// §3.8b — save the current parametrization as a named set.
//
// The set is a PROJECTION of the same deterministic walk that builds the
// §3.10.2 manifest: M_AppendConfig runs exactly as a QUERY_CONFIG would run it,
// and the pager files every capability of the requested ConfigKind as a
// (Scope, WriteKey) record. There is no second enumeration of "what this
// station's configuration consists of" to drift from the first (§1.1 O9).
//
// Kind selects which of the two kinds of set this is: STATION_CFG for a station
// set (deployment data), PAR_CFG for a model set (one model's recipe data).
METHOD SaveConfigSet : BOOL
VAR_INPUT
    SetName : STRING(80);
    Kind    : E_ConfigKind;
END_VAR
VAR
    info    : ST_ConfigSetInfo;
    records : INT;
END_VAR
SaveConfigSet := FALSE;
ConfigPersist.LastSetName := SetName;
ConfigPersist.LastSetRecords := 0;
IF NOT _M_SetOpAllowed() THEN
    RETURN;
END_IF
IF SetName = '' THEN
    RETURN;
END_IF
info.Used := TRUE;
info.SetName := SetName;
info.RootIdentity := Status.Name;
info.SetSchema := CONFIG_SET_SCHEMA;
info.ConfigRev := ConfigRev;
info.Kind := Kind;
IF Kind = E_ConfigKind.PAR_CFG THEN
    info.ModelCode := Model.ModelCode;     // a model set belongs to ONE model
ELSE
    info.ModelCode := '';
END_IF
info.RecordCount := 0;
info.CreatedAt := F_Now();
info.TimeSynchronized := F_TimeSynchronized();
IF NOT _configPager.M_SetupSetSave(Store := _configStore, Info := info) THEN
    RETURN;
END_IF
M_AppendConfig(Pager := _configPager);     // the SAME walk as the manifest
SaveConfigSet := _configPager.M_FinishSetSave(Records => records);
ConfigPersist.LastSetRecords := records;
IF SaveConfigSet THEN
    // The set now lives in the store's retained memory, which is not durable
    // until it is written out - the same promise as any other accepted write.
    _M_MarkPersistPending();
END_IF
END_METHOD

// §3.8b — apply a named set. STAGED and ALL-OR-NOTHING.
//
// Pass 1 validates every record through its owning module's typed handler and
// changes nothing. Only if all of them pass does pass 2 apply them. A
// half-applied machine parametrization is never a valid outcome, and the only
// way to guarantee that is to know the answer for every record before touching
// the first one.
//
// A record whose capability no longer exists fails pass 1 like any other and is
// REPORTED by name - never silently dropped, because a set that quietly skipped
// the one value that mattered restores a machine to almost its commissioned
// state, which is the failure that is hardest to notice.
METHOD LoadConfigSet : BOOL
VAR_INPUT
    SetName : STRING(80);
END_VAR
VAR
    info    : ST_ConfigSetInfo;
    record  : ST_ConfigRecord;
    i       : INT;
    applied : BOOL;
END_VAR
LoadConfigSet := FALSE;
ConfigPersist.LastSetName := SetName;
ConfigPersist.LastSetRecords := 0;
ConfigPersist.LastRejectScope := '';
ConfigPersist.LastRejectKey := '';
IF NOT _M_SetOpAllowed() THEN
    RETURN;
END_IF
IF NOT _configStore.M_ReadInfo(SetName := SetName, Info := info) THEN
    _M_RejectConfigSet(Scope := '', Key := SetName);
    RETURN;
END_IF
IF info.RootIdentity <> Status.Name THEN
    // The set carries the identity of the root that produced it precisely so
    // this can be asked. Every record's Scope is prefixed by that identity, so
    // a mismatch would fail record by record anyway - naming the root instead
    // tells the operator WHY in one line.
    _M_RejectConfigSet(Scope := info.RootIdentity, Key := '');
    RETURN;
END_IF
IF info.Kind = E_ConfigKind.PAR_CFG THEN
    // §3.8b: a MODEL set "shall be applied through the §3.8 changeover
    // transaction (PrepareRecipe -> recursive readiness -> infallible
    // CommitRecipe), never as a sequence of per-field writes". Applying it here
    // would be exactly that forbidden sequence, so it is refused. Saving a
    // model set is supported; loading one is a changeover this build does not
    // implement, and refusing is the honest half of that.
    _M_RejectConfigSet(Scope := info.ModelCode, Key := '');
    RETURN;
END_IF
// ---- pass 1: stage. Nothing in the machine changes in this loop. ----
FOR i := 1 TO info.RecordCount DO
    IF NOT _configStore.M_ReadRecord(SetName := SetName, Index := i,
            Record := record) THEN
        _M_RejectConfigSet(Scope := '', Key := SetName);
        RETURN;
    END_IF
    // §3.8d(e) - CONFIG_SET alone cannot replace a value this session could
    // not edit one at a time. Checked in the staging pass, so nothing moved.
    IF NOT Access.M_PermitsLevelLogged(Required := _M_DataLevelOf(TargetPath := record.Scope,
            WriteKey := record.WriteKey, ForWrite := TRUE)) THEN
        _M_RejectConfigSet(Scope := record.Scope, Key := record.WriteKey);
        RETURN;
    END_IF
    IF NOT _M_StageOneRecord(Record := record) THEN
        _M_RejectConfigSet(Scope := record.Scope, Key := record.WriteKey);
        RETURN;
    END_IF
END_FOR
// ---- pass 2: apply. Every record already proved acceptable on the SAME
// validator, so a refusal here cannot be a data problem. ----
FOR i := 1 TO info.RecordCount DO
    IF NOT _configStore.M_ReadRecord(SetName := SetName, Index := i,
            Record := record) THEN
        _M_ConfigSetHalfApplied(Scope := record.Scope, Key := record.WriteKey);
        RETURN;
    END_IF
    applied := _M_WriteBaseConfig(TargetPath := record.Scope,
        WriteKey := record.WriteKey, Revision := record.Revision,
        TextValue := record.ValueText, Commit := TRUE);
    IF NOT applied THEN
        applied := M_ApplyConfigWrite(Scope := record.Scope,
            WriteKey := record.WriteKey, Revision := record.Revision,
            TextValue := record.ValueText,
            RootReady := (_exec = E_ExecState.READY));
    END_IF
    IF NOT applied THEN
        _M_ConfigSetHalfApplied(Scope := record.Scope, Key := record.WriteKey);
        RETURN;
    END_IF
END_FOR
ConfigRev := ConfigRev + 1;
ConfigPersist.LastSetRecords := info.RecordCount;
_M_MarkPersistPending();
_M_RaiseMaintenance(Reason := E_Reason.EVENT_CONFIG_SET_APPLIED,
    Text := 'std.audit.configSetApplied');
LoadConfigSet := TRUE;
END_METHOD

// §3.8b — would this record be accepted? The same two-step the write path
// takes: framework-owned keys first, then the recursive walk to the owning
// module. Sharing the writers' own code with Commit := FALSE is what makes
// "staged" mean something: a separate validator could pass a record the write
// path would then refuse, and the load would be half-applied after all.
METHOD PRIVATE _M_StageOneRecord : BOOL
VAR_INPUT
    Record : ST_ConfigRecord;
END_VAR
_M_StageOneRecord := _M_WriteBaseConfig(TargetPath := Record.Scope,
    WriteKey := Record.WriteKey, Revision := Record.Revision,
    TextValue := Record.ValueText, Commit := FALSE);
IF _M_StageOneRecord THEN
    RETURN;
END_IF
_M_StageOneRecord := M_StageConfigWrite(Scope := Record.Scope,
    WriteKey := Record.WriteKey, Revision := Record.Revision,
    TextValue := Record.ValueText,
    RootReady := (_exec = E_ExecState.READY));
END_METHOD

// §3.8b — a record passed staging and then failed to apply. This cannot
// happen: both run the same validator on the same data in the same scan. If it
// ever does, the machine is half-parametrized and that is a state the standard
// says is never valid - so it is escalated as a BLOCKING alarm rather than
// returned as a FALSE somebody might retry. A framework defect that leaves a
// machine half-configured has to stop it, not inconvenience it.
METHOD PRIVATE _M_ConfigSetHalfApplied
VAR_INPUT
    Scope : STRING(80);
    Key   : STRING(160);
END_VAR
ConfigPersist.LastRejectScope := Scope;
ConfigPersist.LastRejectKey := Key;
AlarmLog.Raise(Reason := E_Reason.CONFIG_SET_REJECTED,
    Text := 'std.error.configSetHalfApplied', Source := Scope,
    Severity := E_Severity.HIGH, Category := E_Category.SYSTEM,
    ResetClass := E_ResetClass.MANUAL_RESET);
END_METHOD

// §3.8b — refresh the published listing of stored sets. Read-only, so it is
// gated on CONFIG_SET without the audited write path: seeing which sets exist
// is not replacing a machine's parametrization.
METHOD ListConfigSets : BOOL
VAR
    i     : INT;
    total : INT;
END_VAR
ListConfigSets := FALSE;
FOR i := 1 TO PL_Fraktal.MAX_CONFIG_SETS DO
    ConfigSets[i].Used := FALSE;
    ConfigSets[i].SetName := '';
    ConfigSets[i].RecordCount := 0;
END_FOR
ConfigSetCount := 0;
IF NOT Access.Permits(Gate := E_GatedAction.CONFIG_SET) THEN
    RETURN;
END_IF
IF _configStore = 0 THEN
    RETURN;
END_IF
total := _configStore.M_Count();
FOR i := 1 TO PL_Fraktal.MAX_CONFIG_SETS DO
    IF i > total THEN
        EXIT;
    END_IF
    IF _configStore.M_InfoAt(Index := i, Info := ConfigSets[i]) THEN
        ConfigSetCount := i;
    END_IF
END_FOR
ListConfigSets := TRUE;
END_METHOD

// §3.8b — serve one line of a set's JSON document. Line 0 is the header and
// 1..RecordCount are the records, so a client pulls a movable document a line
// at a time and no full document buffer ever exists in the PLC - the same
// paging discipline QUERY_CONFIG already uses for the manifest.
//
// This is what makes a set MOVABLE, which is the point of naming sets at all: a
// station's commissioning can leave the controller as text, be reviewed,
// diffed, version-controlled and put on the next machine.
METHOD ExportConfigSetLine : BOOL
VAR_INPUT
    SetName : STRING(80);
    Line    : INT;
END_VAR
VAR
    info   : ST_ConfigSetInfo;
    record : ST_ConfigRecord;
END_VAR
ExportConfigSetLine := FALSE;
ConfigSetDocument := '';
ConfigSetDocumentLine := Line;
ConfigSetDocumentLines := 0;
IF NOT Access.Permits(Gate := E_GatedAction.CONFIG_SET) THEN
    RETURN;
END_IF
IF _configStore = 0 THEN
    RETURN;
END_IF
IF NOT _configStore.M_ReadInfo(SetName := SetName, Info := info) THEN
    RETURN;
END_IF
ConfigSetDocumentLines := info.RecordCount;
IF Line <= 0 THEN
    ConfigSetDocument := _setJson.M_Header(Info := info);
ELSE
    IF NOT _configStore.M_ReadRecord(SetName := SetName, Index := Line,
            Record := record) THEN
        RETURN;
    END_IF
    IF NOT Access.M_PermitsLevel(Required := _M_DataLevelOf(TargetPath := record.Scope,
            WriteKey := record.WriteKey, ForWrite := FALSE)) THEN
        RETURN;                           // §3.8d(e): the export fails, it is not thinned
    END_IF
    ConfigSetDocument := _setJson.M_Record(Record := record);
END_IF
// An empty line means the projection REFUSED to render it rather than shorten
// it, so the export fails here instead of shipping a document with a hole.
ExportConfigSetLine := (ConfigSetDocument <> '');
END_METHOD

// §3.8b — take one line of a set's JSON document back in. A header line opens
// a store save, record lines append to it, and Commit closes it.
//
// Import writes into the STORE, never into the machine. Bringing a document in
// and applying it to the equipment are two decisions, and keeping them apart is
// what lets LoadConfigSet stay staged and all-or-nothing: an imported set is
// validated against THIS machine's capabilities when somebody chooses to load
// it, not silently as it arrives.
//
// Everything here is untrusted input in the fullest sense - hand-edited, from
// another vendor's tool, from another machine - so the line is parsed into a
// typed record and nothing more is assumed about it (§5.6, §14).
METHOD ImportConfigSetLine : BOOL
VAR_INPUT
    Line   : STRING(480);
    Commit : BOOL;
END_VAR
VAR
    info   : ST_ConfigSetInfo;
    record : ST_ConfigRecord;
END_VAR
ImportConfigSetLine := FALSE;
IF NOT _M_SetOpAllowed() THEN
    _importOpen := FALSE;
    RETURN;
END_IF
IF _setJson.M_ParseHeader(Line := Line, Info := info) THEN
    _importOpen := FALSE;
    info.Used := TRUE;
    info.RecordCount := 0;
    IF NOT _configStore.M_SaveBegin(Info := info) THEN
        RETURN;
    END_IF
    _importOpen := TRUE;
    ConfigPersist.LastSetName := info.SetName;
    ImportConfigSetLine := TRUE;
    RETURN;
END_IF
IF NOT _importOpen THEN
    RETURN;                                // a record before its header: refuse
END_IF
IF _setJson.M_ParseRecord(Line := Line, Record := record) THEN
    ImportConfigSetLine := _configStore.M_SaveRecord(Record := record);
    IF NOT ImportConfigSetLine THEN
        _configStore.M_SaveAbort();
        _importOpen := FALSE;
        RETURN;
    END_IF
ELSIF NOT Commit THEN
    // Neither a header nor a record, and not the closing call: the document is
    // not one this build understands. Abort rather than commit a partial set.
    _configStore.M_SaveAbort();
    _importOpen := FALSE;
    RETURN;
END_IF
IF Commit THEN
    ImportConfigSetLine := _configStore.M_SaveCommit();
    _importOpen := FALSE;
    IF ImportConfigSetLine THEN
        _M_MarkPersistPending();
    END_IF
END_IF
END_METHOD

// §3.8b - take part of a set line. A request carries at most 255 characters
// and an exported line may hold 480, so a longer line arrives as pieces:
// More = TRUE holds this piece and waits for the next; the first piece without
// More completes the line, which is then imported exactly like a whole one.
//
// Joined by FB_ConfigSetJson.M_Join, which measures first: a line that would
// exceed its width is refused and the import aborted - never truncated. (Not
// CONCAT/LEN: those stop at 255, which is the very limit being crossed.)
METHOD ImportConfigSetPiece : BOOL
VAR_INPUT
    Piece  : STRING(255);
    More   : BOOL;
    Commit : BOOL;
END_VAR
VAR
    line : STRING(480);
END_VAR
ImportConfigSetPiece := FALSE;
IF NOT _M_SetOpAllowed() THEN
    _importPart := '';
    RETURN;
END_IF
line := _importPart;
IF NOT _setJson.M_Join(Tail := Piece, Line := line) THEN
    _importPart := '';
    IF _importOpen THEN
        _configStore.M_SaveAbort();
        _importOpen := FALSE;
    END_IF
    RETURN;
END_IF
IF More THEN
    _importPart := line;
    ImportConfigSetPiece := TRUE;             // held, not yet imported
    RETURN;
END_IF
_importPart := '';
ImportConfigSetPiece := ImportConfigSetLine(Line := line, Commit := Commit);
END_METHOD

METHOD M_SequenceAskDecision
VAR_INPUT
    Req : ST_DecisionRequest;
END_VAR
_M_AskDecision(Req := Req);
END_METHOD

METHOD M_SequenceAwait : BOOL
VAR_INPUT
    Idx : INT;
    Label : STRING(120);
    Ok : BOOL;
END_VAR
M_SequenceAwait := _M_Await(Idx := Idx, Label := Label, Ok := Ok);
END_METHOD

METHOD M_SequenceClearDecision
IF Decision.Prompt <> '' THEN
    _M_LogDecision(EventKey := 'std.audit.decisionWithdrawn',
        SourcePath := Decision.SourcePath, Option := 0);
END_IF
_M_ClearDecisionState();
END_METHOD

METHOD M_SequenceComplete
IF _mode = E_Mode.CHANGEOVER THEN
    _M_HostEvent(Kind := E_HostEventKind.CHANGEOVER_DONE, PartUid := '',
        Subject := 'Model', Value := Model.ModelCode,
        Verdict := E_Verdict.NONE, ReasonCode := E_Reason.NONE);
END_IF
_M_Complete();
END_METHOD

METHOD M_SequenceCountGood
CountGood();
END_METHOD

METHOD M_SequenceEndOfCycle : BOOL
M_SequenceEndOfCycle := _M_EndOfCycle();
END_METHOD

METHOD M_SequenceFault
VAR_INPUT
    Reason : E_Reason;
    DescriptionKey : STRING(255);
END_VAR
_M_Fault(Reason, DescriptionKey);
END_METHOD

METHOD M_SequencePartProcessed : BOOL
VAR_INPUT
    Verdict : E_Verdict;
    Reason : E_Reason;
END_VAR
M_SequencePartProcessed :=
    _M_PartProcessed(Verdict := Verdict, Reason := Reason);
END_METHOD

METHOD M_SequencePartReceived : BOOL
M_SequencePartReceived := _M_PartReceived();
END_METHOD

METHOD M_SequencePartRecord : BOOL
VAR_INPUT
    RecordName : STRING(64);
    Value : LREAL;
    Minimum : LREAL;
    Maximum : LREAL;
    Target : LREAL;
    EngUnit : STRING(16);
END_VAR
M_SequencePartRecord := _M_PartRecord(RecordName := RecordName,
    Value := Value, Minimum := Minimum, Maximum := Maximum, Target := Target,
    EngUnit := EngUnit);
END_METHOD

METHOD M_SequencePartStarted
_M_PartStarted();
END_METHOD

// §6.8 register an attached chain (idempotent, bounded). Called from
// FB_SequenceBase.M_Attach, never by project code.
METHOD M_SequenceRegister : BOOL
VAR_INPUT
    Seq : I_Sequence;
END_VAR
VAR
    i : INT;
END_VAR
M_SequenceRegister := FALSE;
IF Seq = 0 THEN
    RETURN;
END_IF
FOR i := 1 TO _sequenceCount DO
    IF _sequences[i] = Seq THEN
        M_SequenceRegister := TRUE;        // already attached: Setup ran again
        RETURN;
    END_IF
END_FOR
IF _sequenceCount >= PL_Fraktal.MAX_SEQUENCES THEN
    RETURN;                                // bounded; refused, never silently dropped
END_IF
_sequenceCount := _sequenceCount + 1;
_sequences[_sequenceCount] := Seq;
M_SequenceRegister := TRUE;
END_METHOD

// §6.10 — reset every attached chain's shared transition result once per
// PLC cycle, before _M_Dispatch drives any step action. This is why a project
// never calls M_BeginScan itself, and why an SFC/LD/FBD chart needs no wiring
// to be safe against a stale ADVANCE (O1).
METHOD PROTECTED _M_BeginSequenceScan
VAR
    i : INT;
END_VAR
// §6.12 — close out the legs the previous scan's dispatch stopped recording. A step
// is live exactly while its action keeps calling M_Step, which is the same fact the
// chart draws, so nothing has to be deregistered when a leg finishes. Sweeping legs
// rather than rows makes this ~10 iterations however long the chain is.
FOR i := 0 TO PL_Fraktal.MAX_PARALLEL_BRANCHES DO
    IF (ActiveSteps[i].RowIdx > 0) AND NOT _branchTouched[i] THEN
        // The row keeps how long it ran: the HMI polls too slowly to have timed it.
        SequenceSteps[ActiveSteps[i].RowIdx].LastDuration := ActiveSteps[i].Elapsed;
        ActiveSteps[i].RowIdx := 0;
        ActiveSteps[i].TimedOut := FALSE;
    END_IF
    _branchTouched[i] := FALSE;
END_FOR
FOR i := 1 TO _sequenceCount DO
    IF _sequences[i] <> 0 THEN
        _sequences[i].M_BeginScan();
    END_IF
END_FOR
END_METHOD

// §6.8 - restart every attached chain. The base calls it where a chain can never
// resume (first scan, mode change, abort, abort in error). Whether a fresh run
// command or an operator reset RESTARTS the chain or lets it resume where an
// error stopped it is the project's policy (§6.9(d)), so a project that wants a
// restart there calls this one line from OnCommandStart / OnOperatorReset.
METHOD PROTECTED _M_RestartSequences
VAR
    i : INT;
END_VAR
FOR i := 1 TO _sequenceCount DO
    IF _sequences[i] <> 0 THEN
        _sequences[i].M_Restart();
    END_IF
END_FOR
// A decision belongs to the chain step that asked it; a restarted chain asks again.
Decision.Prompt := '';
DecisionAnswer := 0;
END_METHOD

// §3.14 - an aborted mode chain is abandoned, never resumed: restart every
// attached chain so the next command starts at N000 (§6.8).
METHOD PROTECTED OnAbort : DINT
OnAbort := SUPER^.OnAbort();
_M_RestartSequences();
END_METHOD

// §3.14 - error-state abort abandons the chain the same way (§6.8).
METHOD PROTECTED OnAbortInError : DINT
OnAbortInError := SUPER^.OnAbortInError();
_M_RestartSequences();
END_METHOD

// §6.9(e) — a step said something worth recording that is not a failure.
// Deliberately does NOT touch _exec: no fault is adopted, _M_Dispatch keeps
// running, and the chain follows its own recovery path. The ring entry is
// AUTO_RESET come+gone (§8.3(c)) so it can never block the next Start.
METHOD M_SequenceWarn : BOOL
VAR_INPUT
    Diag : ST_Diagnostic;
END_VAR
VAR
    d    : ST_Diagnostic;
    slot : INT;
END_VAR
d := Diag;
IF d.SourcePath = '' THEN
    d.SourcePath := _name;
END_IF
F_RationalizeDiagnostic(Diag := d);   // §8.8 owns a registered reason's level
IF (_seqIndex >= 1) AND (_seqIndex <= SequenceStepCount) THEN
    SequenceSteps[_seqIndex].WarningActive := TRUE;
    // A message about THIS Unit has nowhere to drill; one about a child keeps the
    // child's path, so the chart links to the module the message is about.
    IF d.SourcePath = _name THEN
        _M_SequenceAnnotate(RowIdx := _seqIndex, IsError := FALSE,
            Key := d.Description, SourcePath := '');
    ELSE
        _M_SequenceAnnotate(RowIdx := _seqIndex, IsError := FALSE,
            Key := d.Description, SourcePath := d.SourcePath);
    END_IF
END_IF
slot := AlarmLog.Raise(Reason := d.ReasonCode, Text := d.Description,
    Source := d.SourcePath, Severity := d.Severity, Category := d.Category,
    ResetClass := E_ResetClass.AUTO_RESET);
IF slot > 0 THEN
    AlarmLog.Gone(Slot := slot);       // an occurrence, not a standing condition
END_IF
M_SequenceWarn := TRUE;
END_METHOD

// §6.9 — a step raised a first-out itself. Stamp the flow-chart row with the
// error and its link before adopting the diagnostic, so the §3.13 chart can mark
// the step red and drill into the module that actually failed even when the step
// passed Awaits := 0. Adopting the diagnostic stops the chain: _M_FaultDiag puts
// the Unit in ERROR and _M_Dispatch no longer runs.
METHOD M_SequenceRaise : BOOL
VAR_INPUT
    Diag     : ST_Diagnostic;
    LinkPath : STRING(255);
END_VAR
M_SequenceRaise := FALSE;
IF (_seqIndex >= 1) AND (_seqIndex <= SequenceStepCount) THEN
    SequenceSteps[_seqIndex].ErrorActive := TRUE;
    _M_SequenceAnnotate(RowIdx := _seqIndex, IsError := TRUE,
        Key := Diag.Description, SourcePath := LinkPath);
END_IF
_M_FaultDiag(Diag := Diag);
M_SequenceRaise := TRUE;
END_METHOD

// §6.9 — the ERROR state ended: clear the flow-chart error marks and re-arm
// every attached chain so the step that raised the fault re-evaluates its
// command. A project writes nothing for this (§1.1 O1).
METHOD PROTECTED _M_ResumeSequencesAfterError
VAR
    i : INT;
END_VAR
FOR i := 1 TO SequenceStepCount DO
    SequenceSteps[i].ErrorActive := FALSE;
END_FOR
_M_SequenceAnnotationClear(RowIdx := 0, IsError := TRUE);
FOR i := 1 TO _sequenceCount DO
    IF _sequences[i] <> 0 THEN
        _sequences[i].M_ResumeAfterError();
    END_IF
END_FOR
END_METHOD

// I_SequenceHost (§6.7/§6.8) — step record for a separately-compiled chain.
METHOD M_SequenceSetStep
VAR_INPUT
    StepNo : INT;
    StepName : STRING(120);
    Awaits : I_Module;
    AwaitingLabel : STRING(120);
    TimeClass : E_TimeClass;
    ExpectedTime : TIME;
    Branch : INT;
END_VAR
// §6.12 — a step on a concurrent LEG publishes its own row and nothing else. The
// Unit's CurrentStep, the §6.9 stall walk and the §8.11.4 profiler are singular by
// definition; letting a leg write them would make the walk report whichever leg
// happened to run last. A leg is timed and guarded on its own row instead, so
// _M_SetStep keeps the signature every inline chain already calls (§1.1 O1).
IF Branch > 0 THEN
    _M_RecordSequenceStep(StepNo := StepNo, StepName := StepName, Awaits := Awaits,
        AwaitingLabel := AwaitingLabel, TimeClass := TimeClass, ExpectedTime := ExpectedTime,
        Branch := Branch);
    RETURN;
END_IF
_M_SetStep(StepNo := StepNo, StepName := StepName,
    Awaits := Awaits, AwaitingLabel := AwaitingLabel, TimeClass := TimeClass,
    ExpectedTime := ExpectedTime);
END_METHOD

METHOD M_SequenceStepGate : BOOL
VAR_INPUT
    Steppable : BOOL;
END_VAR
M_SequenceStepGate := _M_StepGate(Steppable := Steppable);
END_METHOD

// §3.4/§8.11 — accept a pending Stop BETWEEN cycles: the open profile fragment
// (just the wait step) is abandoned, not published as a production cycle.
METHOD M_SequenceStopNow
Profiler.CycleAbandon();
_stopReq := FALSE;
Execute := FALSE;
_M_Complete();
END_METHOD

// §3.4 — a chain polls this at its between-cycles wait step.
METHOD M_SequenceStopPending : BOOL
M_SequenceStopPending := _stopReq AND (_exec = E_ExecState.BUSY);
END_METHOD

METHOD M_SequenceTakeDecision : INT
M_SequenceTakeDecision := _M_TakeDecision();
END_METHOD

// §7.6.1a — single gated entry for a HELD manual action (hold-to-run). Same
// gates as ManualCommandTo: this Unit in MANUAL (§3.4) and MANUAL access
// (§7.7). Held := TRUE latches the request; FALSE releases it immediately.
//
// The release is explicit AND the latch expires, deliberately both: an explicit
// release stops the motion the moment the operator lets go, and the deadline
// stops it when no release ever arrives because the client vanished. Relying on
// either alone leaves one of those two cases moving.
//
// Hold-to-run over a transport is NON-SAFETY (no dead-man, TC3 §7.6): the
// enabling device is the safety-rated fact, derived below from the §9 facet and
// carried to the module, which weighs it itself.
METHOD ManualHeldTo : BOOL
VAR_INPUT
    TargetPath : STRING(255);
    Value      : DINT;
    Held       : BOOL;
END_VAR
VAR
    auditSlot : INT;
END_VAR
ManualHeldTo := FALSE;
IF NOT Held THEN
    // A release is always honoured, whatever the mode or access says now. The
    // operator letting go must never depend on a gate that may have changed
    // since they took hold of it.
    _heldActive := FALSE;
    _heldPath := '';
    _heldValue := 0;
    ManualHeldTo := TRUE;
    RETURN;
END_IF
IF _mode <> E_Mode.MANUAL THEN
    auditSlot := AlarmLog.Raise(Reason := E_Reason.NONE,
        Text := 'std.audit.manualCommandWrongMode', Source := TargetPath,
        Severity := E_Severity.LOW, Category := E_Category.SYSTEM,
        ResetClass := E_ResetClass.AUTO_RESET);
    IF auditSlot > 0 THEN AlarmLog.Gone(Slot := auditSlot); END_IF
    RETURN;
END_IF
IF NOT Access.PermitsLogged(Gate := E_GatedAction.MANUAL) THEN
    RETURN;                              // §7.7 denial already audited
END_IF
// Prove the target accepts it BEFORE latching, so a hold on a module that
// refuses never becomes a standing request nobody can see the source of.
IF NOT _M_RouteHeld(TargetPath := TargetPath, Value := Value) THEN
    RETURN;
END_IF
_heldPath := TargetPath;
_heldValue := Value;
_heldActive := TRUE;
_heldSinceMs := TIME_TO_DWORD(TIME());
ManualHeldTo := TRUE;
END_METHOD

// §7.6.1a — derive the enabling-device fact from THIS root's §9 safety facet and
// carry it to the owning module through the registered-child walk.
//
// F_ManualEnable is the single place the fact is derived, so grepping for it
// lists every path by which motion is authorised by an enabling device. Until
// now it had no production caller at all - the capability existed and nothing
// reached it.
METHOD PROTECTED _M_RouteHeld : BOOL
VAR_INPUT
    TargetPath : STRING(255);
    Value      : DINT;
END_VAR
VAR
    enable : ST_ManualEnableStatus;
END_VAR
enable := F_ManualEnable(Safety := Safety);
_M_RouteHeld := M_ApplyHeld(Scope := TargetPath, Value := Value,
    Enable := enable);
END_METHOD

// §3.13/§3.10.2 — raise the manifest revision ONCE the flow chart has stopped
// growing, rather than once per row discovered.
//
// The rows are the manifest's largest and most volatile contributor and they
// appear one at a time as the chain visits them, so a per-row bump turned one
// mode entry into one full-manifest refetch per step. This waits for the burst
// to settle and then charges for it once.
//
// The delay is bounded and small (PL_Fraktal.CHART_REV_SETTLE_MS): the chart
// appears fractionally later and COMPLETE, instead of promptly and then being
// refetched fourteen more times.
METHOD PRIVATE _M_ChartRevCyclic
VAR
    elapsed : DWORD;
END_VAR
IF NOT _chartDirty THEN
    RETURN;
END_IF
// Unsigned subtraction, so the monotonic counter wrapping cannot fabricate a
// settled chart (TC3 §8.11).
elapsed := TIME_TO_DWORD(TIME()) - _chartTouchedMs;
IF elapsed < PL_Fraktal.CHART_REV_SETTLE_MS THEN
    RETURN;                            // still growing: let the burst finish
END_IF
_chartDirty := FALSE;
ConfigRev := ConfigRev + 1;
END_METHOD

// §7.6.1a — re-assert the latched hold every scan, and drop it when the client
// stops refreshing. The module's own freshness timer stops the motion; this
// stops the ROOT from going on asking for it.
METHOD PRIVATE _M_HeldCyclic
VAR
    elapsed : DWORD;
END_VAR
IF NOT _heldActive THEN
    RETURN;
END_IF
// Leaving MANUAL, or losing the access that granted it, ends the hold at once.
IF _mode <> E_Mode.MANUAL THEN
    _heldActive := FALSE;
    RETURN;
END_IF
IF NOT Access.Permits(Gate := E_GatedAction.MANUAL) THEN
    _heldActive := FALSE;
    RETURN;
END_IF
// Unsigned subtraction, so the monotonic counter wrapping cannot fabricate an
// expired hold (TC3 §8.11).
elapsed := TIME_TO_DWORD(TIME()) - _heldSinceMs;
IF elapsed > PL_Fraktal.MANUAL_HELD_REFRESH_MS THEN
    _heldActive := FALSE;                // client went quiet: let go for it
    RETURN;
END_IF
_M_RouteHeld(TargetPath := _heldPath, Value := _heldValue);
END_METHOD

// §7.6.1 — single gated manual-command entry for the HMI. Accepts ONLY when this
// Unit is in MANUAL (§3.4) AND the user holds MANUAL access (§7.7). Routes to the
// target module's ManualCommand (through the command surface — defended, not
// bypassed). Logs every accept/reject as a §8.3 event. Concrete Units override
// _M_RouteManual to map TargetPath -> the child module.
METHOD ManualCommandTo : BOOL
VAR_INPUT
    TargetPath : STRING(255);
    Value : DINT;
END_VAR
VAR
    auditSlot : INT;
END_VAR
ManualCommandTo := FALSE;
IF _mode <> E_Mode.MANUAL THEN
    auditSlot := AlarmLog.Raise(Reason := E_Reason.NONE,
        Text := 'std.audit.manualCommandWrongMode', Source := TargetPath,
        Severity := E_Severity.LOW, Category := E_Category.SYSTEM, ResetClass := E_ResetClass.AUTO_RESET);
    IF auditSlot > 0 THEN AlarmLog.Gone(Slot := auditSlot); END_IF
    RETURN;
END_IF
IF NOT Access.PermitsLogged(Gate := E_GatedAction.MANUAL) THEN
    RETURN;                              // §7.7 denial already audited
END_IF
ManualCommandTo := _M_RouteManual(TargetPath := TargetPath, Value := Value);
IF ManualCommandTo THEN
    auditSlot := AlarmLog.Raise(Reason := E_Reason.NONE,
        Text := 'std.audit.manualCommandAccepted', Source := TargetPath,
        Severity := E_Severity.LOW, Category := E_Category.SYSTEM, ResetClass := E_ResetClass.AUTO_RESET);
ELSE
    auditSlot := AlarmLog.Raise(Reason := E_Reason.UNSUPPORTED_COMMAND,
        Text := 'std.audit.manualCommandRejected', Source := TargetPath,
        Severity := E_Severity.LOW, Category := E_Category.SYSTEM, ResetClass := E_ResetClass.AUTO_RESET);
END_IF
IF auditSlot > 0 THEN AlarmLog.Gone(Slot := auditSlot); END_IF
END_METHOD

PROPERTY ModeActive : E_Mode
GET
ModeActive := _mode;
END_GET
END_PROPERTY

PROPERTY ModelCode : STRING(64)
GET
ModelCode := Model.ModelCode;
END_GET
END_PROPERTY

PROPERTY ModuleType : E_ModuleType
GET
ModuleType := E_ModuleType.UNIT;
END_GET
END_PROPERTY

// base first (§3.14.2); then children, one-shot init, mode transition, stall watch
METHOD PROTECTED OnCyclic : DINT
VAR
    publishIdx : INT;
    modeIdx    : E_Mode;
    styleIdx   : E_RunStyle;
    previousMode : E_Mode;
    modeExitResult : DINT;
    highestSeverity : E_Severity;
    alarmActive : BOOL;
    heldReported : BOOL;
END_VAR
OnCyclic := SUPER^.OnCyclic();
_M_BeginSequenceScan();                               // §6.10 one-scan result reset for every attached chain
_M_TickChildren();
IF _pLine <> 0 THEN
    IF _lineHost THEN
        _pLine^.Cyclic();                             // §3.8e the hosting root runs the line
    END_IF
    // A line value can change without a write through THIS root: a mirror applies
    // its owner's revision, a second root on the line edits it. Either way this
    // root's manifest now reads differently, so its revision moves.
    IF _pLine^.OutImm.Revision <> _lineRevSeen THEN
        _lineRevSeen := _pLine^.OutImm.Revision;
        ConfigRev := ConfigRev + 1;
    END_IF
END_IF
_M_OeeUpdate();                                       // §8.5.1 time accounting + sampling
M_ShiftTick(Now := F_Now(), Synchronized := F_TimeSynchronized());   // §8.5.2
AlarmLog.Cyclic();                                    // §8.10 shelf auto-expiry
_M_EngineeringCyclic();                               // §7.5.2 standing gate annunciation
_healthPublisher.Cyclic(Input := _healthInput, ParCfg := _healthParCfg,
    Configured := _healthConfigured);                 // §2.7/§8.12 alarm edges + values
SystemHealth := _healthPublisher.Status;
_M_ChartRevCyclic();                                  // §3.13 coalesced chart revision
_M_HeldCyclic();                                      // §7.6.1a hold-to-run re-assert
_M_ConfigPersistCyclic();                             // §3.8b durability window
_M_DrainRestoreLoss();                                // §3.8b restore annunciation
_M_HandleHmiRequest();                                // §3.10 request mailbox
_M_DecisionCyclic();                                  // §6.11 timeout/default/overlap resolver
Access.Cyclic();
alarmActive := _M_HighestSeverity(Highest := highestSeverity);
_towerMapper.Cyclic(MachineState := MachineState, AlarmActive := alarmActive,
    HighestSeverity := highestSeverity,
    OperatorActionRequired := (Decision.Prompt <> ''),
    LampTestRequest := _lampTestRequest, ParCfg := _towerParCfg);
_lampTestRequest := FALSE;
SignalTower := _towerMapper.Status;
// §9.8 data-driven Control On/Off request endpoint. Off wins if both arrive;
// the domain/power-group implementation still validates safety, health and rearm.
ControlOnRequest := FALSE;
ControlOffRequest := FALSE;
IF ReqControlOff THEN
    ReqControlOff := FALSE;
    ReqControlOn := FALSE;
    IF Access.PermitsLogged(Gate := E_GatedAction.POWER_CONTROL) THEN
        ControlOffRequest := TRUE;
    END_IF
ELSIF ReqControlOn THEN
    ReqControlOn := FALSE;
    IF Access.PermitsLogged(Gate := E_GatedAction.POWER_CONTROL) THEN
        ControlOnRequest := TRUE;
    END_IF
END_IF
// §3.14.4 — pending mode change; §3.4.1 style decides graceful vs immediate
IF _modePend THEN
    IF _exec = E_ExecState.BUSY THEN
        IF ModePolicy[TO_INT(_mode)].Style = E_ModeSwitchStyle.GRACEFUL THEN
            _stopReq := TRUE;                             // finish the cycle at its stop point
        ELSE
            modeExitResult := OnModeExit(FirstCall := _modeExitFirst,
                RequestedMode := _modeReq);
            _modeExitFirst := FALSE;
            IF modeExitResult = 0 THEN
                OnAbort();                                // IMMEDIATE: cancel now (override may defer)
            END_IF
        END_IF
    ELSE
        IF _exec <> E_ExecState.READY THEN
            Execute := FALSE;                             // release the run command (§6.1 reset)
        ELSE
            previousMode := _mode;
            _mode := _modeReq;
            _modePend := FALSE;
            _modeExitFirst := FALSE;
            _M_CascadeMode(_mode);                        // §3.7 cascade [TC3]
            OnModeChanged(NewMode := _mode, OldMode := previousMode);
        END_IF
    END_IF
END_IF
// §8.3(c) — automatic fault capture: ERROR entry raises, ERROR exit marks gone
IF (_exec = E_ExecState.ERROR) AND (_faultEvt = 0) THEN
    _faultEvt := AlarmLog.RaiseDiag(D := _diag, ResetClass := E_ResetClass.MANUAL_RESET);
    _M_PartAborted();                  // §3.16.3: a faulted part leaves without a valid result
ELSIF (_exec <> E_ExecState.ERROR) AND (_faultEvt > 0) THEN
    AlarmLog.Gone(Slot := _faultEvt);                            // -> WAIT_RESET (blocking)
    _faultEvt := 0;
END_IF
// §6.9 — instant rollup on awaited Error; adopt a HELD child; stall as PENDING otherwise
IF _exec = E_ExecState.BUSY THEN
    IF (_awaits <> 0) AND_THEN _awaits.FaultActive THEN
        _M_FaultDiag(_awaits.GetFaultSummary());
    ELSE
        // §6.1 HELD — the held module is waiting on a condition it can name, so
        // report THAT instead of letting StallTime expire into a generic stall. A
        // declared wait is not a stall, so the watchdog stays disarmed while it lasts.
        //
        // The hold rolls up whether or not the step awaits the child (§1.1 O1: the
        // project must not have to remember a call to stay correct). `Awaits := 0`
        // says "this step owns the child's FAULT disposition" (§6.9, press AUTO
        // N200 offering scrap/return) - it does not say "stay silent while the ram
        // is HELD". A hold is recoverable information that clears itself and never
        // blocks a restart, so suppressing it only produced a Unit that sat BUSY
        // with an empty diagnostic while its own child correctly reported Held.
        // Prefer the awaited module: when a step named one it is the most specific
        // source. _M_RollupHold is called on exactly the scans the awaited branch
        // did not fire, because TwinCAT does not short-circuit and calling both
        // would let a second held child overwrite the named one.
        heldReported := FALSE;
        IF (_awaits <> 0) AND_THEN _awaits.HoldActive THEN
            _M_HoldDiag(Diag := _awaits.GetFaultSummary());
            heldReported := TRUE;
        ELSE
            heldReported := _M_RollupHold();   // §8.2 first held registered child
        END_IF
        IF heldReported THEN
            _tStall(IN := FALSE);
        ELSE
            IF Held THEN
                _M_ClearPending();     // the hold ended: drop any stall text it outlived
            END_IF
            _tStall(IN := TRUE, PT := SEL(CurrentStep.ExpectedTime > T#0S, StallTime, CurrentStep.ExpectedTime));
            IF _tStall.Q THEN
                _M_StallWalk();
            END_IF
        END_IF
    END_IF
ELSE
    _tStall(IN := FALSE);
END_IF
// §6.9(a) — every new fault joins the shift-change ring, no historian needed
_fTrig(CLK := (_exec = E_ExecState.ERROR));
_errClr(CLK := (_exec <> E_ExecState.ERROR));
IF _errClr.Q THEN
    _M_ResumeSequencesAfterError();   // §6.9 re-evaluate, do not resume blind
END_IF
IF _fTrig.Q THEN
    _M_PushHistory(_diag);
END_IF
// §8.11.4(d) — creeping WORK time is a MAINTENANCE event (Low), not downtime:
// the profiler pulses once per excursion past the configured baseline band.
IF Profiler.DegradedTrig THEN
    _M_RaiseMaintenance(Reason := E_Reason.CYCLE_TIME_DEGRADED,
        Text := 'std.maintenance.cycleTimeDegraded');
END_IF
ModeActivePublished := _mode;
RunningPublished := (_exec = E_ExecState.BUSY);
StopPendingPublished := _stopReq AND (_exec = E_ExecState.BUSY);
FOR publishIdx := 0 TO PL_Fraktal.MODE_COUNT - 1 DO
    modeIdx := publishIdx;
    SupportedModesPublished[publishIdx] := _M_Supports(Mode := modeIdx);
END_FOR
FOR publishIdx := 0 TO 2 DO
    styleIdx := publishIdx;
    SupportedRunStylesPublished[publishIdx] := _M_SupportsRunStyle(Style := styleIdx);
END_FOR
END_METHOD

// §8.13 — derive the tower input from the authoritative active-event table.
METHOD PRIVATE _M_HighestSeverity : BOOL
VAR_IN_OUT
    Highest : E_Severity;
END_VAR
VAR
    i : INT;
END_VAR
_M_HighestSeverity := FALSE;
Highest := E_Severity.LOW;
FOR i := 1 TO PL_Fraktal.MAX_ALARM_ACTIVE DO
    IF AlarmLog.Active[i].State <> E_AlarmState.CLOSED THEN
        IF NOT _M_HighestSeverity OR (AlarmLog.Active[i].Severity > Highest) THEN
            Highest := AlarmLog.Active[i].Severity;
        ELSE
            ;
        END_IF
        _M_HighestSeverity := TRUE;
    ELSE
        ;
    END_IF
END_FOR
END_METHOD

// §8.13 — remote request is MANUAL-gated and starts only while the Unit is idle.
METHOD RequestLampTest : BOOL
RequestLampTest := FALSE;
IF _exec = E_ExecState.BUSY THEN
    RETURN;
END_IF
IF NOT Access.PermitsLogged(Gate := E_GatedAction.MANUAL) THEN
    RETURN;
END_IF
_lampTestRequest := TRUE;
RequestLampTest := TRUE;
END_METHOD

// Startup station-convention seam. Runtime config writes require a registered
// typed capability; this method is not published by OPC UA.
METHOD SetSignalTowerConfig : BOOL
VAR_INPUT
    ParCfg : ST_SignalTowerParCfg;
END_VAR
IF (ParCfg.SchemaVersion <> 1) OR (ParCfg.LampTestDuration <= T#0S) THEN
    SetSignalTowerConfig := FALSE;
    RETURN;
END_IF
_towerParCfg := ParCfg;
SetSignalTowerConfig := TRUE;
END_METHOD

// TC3/platform adapter injection. Raw probe values remain OPC-UA-hidden; the
// health publisher validates and republishes the bounded status surface.
METHOD SetSystemHealth : BOOL
VAR_INPUT
    Input  : ST_SystemHealthInput;
    ParCfg : ST_SystemHealthParCfg;
END_VAR
IF ParCfg.SchemaVersion <> 1 THEN
    SetSystemHealth := FALSE;
    RETURN;
END_IF
_healthInput := Input;
_healthParCfg := ParCfg;
_healthConfigured := TRUE;
SetSystemHealth := TRUE;
END_METHOD

// §3.14 hook — one-shot after first operational scan
METHOD PROTECTED OnInit : DINT
VAR
    i : INT;
END_VAR
OnInit := SUPER^.OnInit();
_M_RestartSequences();         // §6.8 every attached chain starts at N000
SequenceViewEnabled := TRUE;   // §3.13 a Unit has a chain worth drawing;
                               // a concrete Unit may vary this per mode
Access.Setup(Provider := 0, pAlarmLog := ADR(AlarmLog)); // preserves an injected provider
_healthPublisher.Setup(SourcePath := CONCAT(Status.Name, '.SystemHealth'),
    pAlarmLog := ADR(AlarmLog));
// §3.10.2 — seed the manifest revision from boot time so every PLC restart or
// re-activation yields a NEW value (a plain counter would repeat after reboot
// and an HMI could keep a stale manifest undetected). Config writes increment.
ConfigRev := DT_TO_UDINT(F_Now());
// §3.8b — the durability provider defaults to the shipped LOCAL_RETAIN writer.
// SetConfigPersistence may already have replaced it, so this never overwrites an
// injected one.
IF _persistence = 0 THEN
    _persistence := _persistWriter;
END_IF
// The framework's OWN station config is subject to the same rule it imposes on
// every module: version 0 is a first boot that lost nothing, any other
// unrecognized version means a real ModePolicy image was rejected and that is
// annunciated with this root's path. The base used to treat both cases as a
// silent re-initialize, which is exactly the "runs on defaults while presenting
// itself as commissioned" failure §3.8b exists to prevent.
IF NOT M_RestoreStationCfg(pVersion := ADR(_modePolicyVersion),
        SchemaVersion := MODE_POLICY_SCHEMA) THEN
    _M_InitModePolicy();
    FOR i := 0 TO PL_Fraktal.MODE_COUNT - 1 DO
        _modePolicyStored[i] := ModePolicy[i];
    END_FOR
ELSE
    FOR i := 0 TO PL_Fraktal.MODE_COUNT - 1 DO
        ModePolicy[i] := _modePolicyStored[i];
    END_FOR
END_IF
END_METHOD

// §3.14 hook — after the new mode is committed
METHOD PROTECTED OnModeChanged : DINT
VAR_INPUT
    NewMode : E_Mode;
    OldMode : E_Mode;
END_VAR
_M_HostEvent(Kind := E_HostEventKind.MODE_CHANGED, PartUid := '',
    Subject := 'Mode', Value := TO_STRING(TO_DINT(NewMode)),
    Verdict := E_Verdict.NONE, ReasonCode := E_Reason.NONE);
// §3.13 — the chart belongs to the mode that is running. A project writes nothing
// for this: it lands in the base hook every override calls SUPER^ on first (§3.14.2).
_M_ResetSequenceRows();
// §6.8 — and so do the chains: a new mode starts every chain at N000.
_M_RestartSequences();
OnModeChanged := 0;
END_METHOD

// Core §11.6: CHANGEOVER starts when its guided sequence actually starts, not
// merely when the operator selects the mode or transactionally loads a model.
METHOD PROTECTED OnCommandStart : DINT
OnCommandStart := SUPER^.OnCommandStart();
IF _mode = E_Mode.CHANGEOVER THEN
    _M_HostEvent(Kind := E_HostEventKind.CHANGEOVER_STARTED, PartUid := '',
        Subject := 'Model', Value := Model.ModelCode,
        Verdict := E_Verdict.NONE, ReasonCode := E_Reason.NONE);
END_IF
END_METHOD

// §3.14.4 — called every scan while a mode request is pending and the Unit is BUSY.
// Return 0 = consent to immediate cancel (default); >0 = still stopping gracefully.
METHOD PROTECTED OnModeExit : DINT
VAR_INPUT
    FirstCall : BOOL;
    RequestedMode : E_Mode;
END_VAR
OnModeExit := 0;
END_METHOD

// §8.3(b) — deliberate operator reset of blocking events (release-gated per §7.6/§14).
// ONE operator action has to make the Unit restartable, so this closes the blocking
// events AND clears the latched control state they were reporting: see _M_RecoverState.
METHOD OperatorReset : BOOL
IF NOT Access.PermitsLogged(Gate := E_GatedAction.ALARM_RESET) THEN
    OperatorReset := FALSE;            // §7.7
    RETURN;
END_IF
OperatorReset := _M_RecoverState();
OperatorReset := AlarmLog.OperatorReset() OR OperatorReset;
END_METHOD

// §8.3(b)/§6.1 — the control-state half of a reset. Closing the alarm alone left the
// machine locked: the Unit's run command and the child commands its mode chain had
// issued both stayed asserted, and §6.1's Execute-drop reset — the only exit from a
// latched terminal state — needs them LOW. A frozen chain cannot drop them itself,
// because a Unit that is not BUSY never calls _M_Dispatch again, so the step holding
// `child.Execute := TRUE` never runs. Nothing else in the system clears it, and the
// next Start re-issues the same already-TRUE input: no rising edge, the child stays
// in ERROR, and the Unit re-adopts the fault through the §8.2 rollup. That is the
// press hard-lock. Returns TRUE when there was something to recover.
// Deliberately does NOT clear ERROR here: Cyclic keeps that ownership (§6.1), so a
// cause that is still live re-faults on the next command edge instead of vanishing.
METHOD PROTECTED _M_RecoverState : BOOL
_M_RecoverState := FALSE;
IF (_exec <> E_ExecState.ERROR) AND NOT AlarmLog.Blocking THEN
    RETURN;                            // nothing latched: a stray reset changes nothing
END_IF
OnOperatorReset();                     // §3.14 hook: withdraw outputs, reset mode chains
_M_ReleaseChildCommands();             // stranded child commands -> READY next scan
_M_ClearPending();
_stopReq := FALSE;
IF _exec = E_ExecState.BUSY THEN
    // Defined safe reaction (§5.6) for a blocking event raised by application code
    // while the mode chain still runs: a recovery reset cancels what was running
    // rather than leaving a chain we just reset still driving the machine.
    AbortCommand();
END_IF
Execute  := FALSE;                     // stale run command -> Unit READY next scan
_faultEvt := 0;                        // the event is closed here, not by a later Gone()
_M_RecoverState := TRUE;
END_METHOD

// §3.14 hook — an accepted operator reset is recovering this Unit. Override to
// withdraw application outputs and reset application-owned mode chains before the
// base releases the run command; call SUPER^.OnOperatorReset() first (§3.14.2).
// Called only when something was actually latched (ERROR or a blocking alarm), so an
// override may assume it is a recovery, not a routine poll.
METHOD PROTECTED OnOperatorReset : DINT
OnOperatorReset := 0;
END_METHOD

// Application-only seam for an ordinary hardwired fault-reset/acknowledge button,
// mirroring RequestLocalControl (§9.8): it is a METHOD, not OPC UA data, so remote
// clients still go through the access-gated OPERATOR_RESET request and cannot reach
// this path. A cabinet button IS its own authorization (physical presence), so it
// carries no §7.7 session check — but the reset is still audited as a §8.3 event,
// and it recovers exactly the same state as an operator reset, never more.
// The composition root calls this from its hardware driver on the button's rising
// edge, once per root Unit it should clear.
METHOD RequestLocalReset : BOOL
VAR
    auditSlot : INT;
END_VAR
auditSlot := AlarmLog.Raise(Reason := E_Reason.NONE,
    Text := 'std.audit.localResetRequested', Source := _name,
    Severity := E_Severity.LOW, Category := E_Category.SYSTEM,
    ResetClass := E_ResetClass.AUTO_RESET);
IF auditSlot > 0 THEN AlarmLog.Gone(Slot := auditSlot); END_IF
RequestLocalReset := _M_RecoverState();
RequestLocalReset := AlarmLog.OperatorReset() OR RequestLocalReset;
END_METHOD

// §3.8 optional HMI/MES selection catalog. Recipe providers remain pluggable;
// the application registers only the model identities it deliberately exposes.
METHOD RegisterAvailableModel : BOOL
VAR_INPUT
    Id : ST_ModelId;
END_VAR
VAR
    i : INT;
END_VAR
RegisterAvailableModel := FALSE;
IF (Id.ModelCode = '') OR (AvailableModelCount >= PL_Fraktal.MAX_RECIPES) THEN
    RETURN;
END_IF
FOR i := 1 TO AvailableModelCount DO
    IF AvailableModels[i].ModelCode = Id.ModelCode THEN
        RETURN;
    END_IF
END_FOR
AvailableModelCount := AvailableModelCount + 1;
AvailableModels[AvailableModelCount] := Id;
ConfigRev := ConfigRev + 1;    // §3.10.2 — manifest changed
RegisterAvailableModel := TRUE;
END_METHOD

// §9.8 remote control-domain request. The acknowledgement is the result of this
// authorization check; it is never reported accepted before POWER_CONTROL runs.
METHOD RequestControlPower : BOOL
VAR_INPUT
    ControlOn : BOOL;
END_VAR
RequestControlPower := FALSE;
IF NOT Access.PermitsLogged(Gate := E_GatedAction.POWER_CONTROL) THEN
    RETURN;
END_IF
IF ControlOn THEN
    ReqControlOn := TRUE;
    ReqControlOff := FALSE;
ELSE
    ReqControlOff := TRUE;                         // Off wins if both were requested
    ReqControlOn := FALSE;
END_IF
RequestControlPower := TRUE;
END_METHOD

// §6.11 authoritative decision entry. START_STOP is the access gate because the
// answer advances a running Unit chain; option-specific process releases append
// through _M_AppendDecisionInterlocks. A stale/invalid answer never latches.
METHOD SubmitDecision : BOOL
VAR_INPUT
    Option : INT;
END_VAR
VAR_IN_OUT
    Report : ST_ReleaseReport;
END_VAR
Report.Count := 0;
Report.Released := FALSE;
SubmitDecision := FALSE;
IF NOT Access.PermitsLogged(Gate := E_GatedAction.START_STOP) THEN
    _M_AddReason(Report := Report, Text := 'std.release.insufficientStartStop',
        Reason := E_Reason.NONE, Kind := E_ReleaseKind.ACCESS);
END_IF
IF (_exec <> E_ExecState.BUSY) OR (Decision.Prompt = '') THEN
    _M_AddReason(Report := Report, Text := 'std.release.noActiveDecision',
        Reason := E_Reason.NONE, Kind := E_ReleaseKind.OTHER);
ELSIF (Option < 1) OR (Option > PL_Fraktal.MAX_OPTIONS) THEN
    _M_AddReason(Report := Report, Text := 'std.release.invalidDecisionOption',
        Reason := E_Reason.UNSUPPORTED_COMMAND, Kind := E_ReleaseKind.OTHER);
ELSIF Decision.Options[Option] = '' THEN
    _M_AddReason(Report := Report, Text := 'std.release.invalidDecisionOption',
        Reason := E_Reason.UNSUPPORTED_COMMAND, Kind := E_ReleaseKind.OTHER);
ELSE
    _M_AppendDecisionInterlocks(Option := Option, Report := Report);
END_IF
Report.Released := (Report.Count = 0);
IF Report.Released THEN
    DecisionAnswer := Option;
    SubmitDecision := TRUE;
END_IF
END_METHOD

// §7.7 persistent per-root policy edit. The policy's own ACCESS_POLICY threshold
// is rechecked before any threshold — including itself — can change.
METHOD SetAccessLevel : BOOL
VAR_INPUT
    Gate : E_GatedAction;
    Level : E_AccessLevel;
END_VAR
SetAccessLevel := FALSE;
IF NOT Access.PermitsLogged(Gate := E_GatedAction.ACCESS_POLICY) THEN
    RETURN;
END_IF
// Never allow an anonymous/lower session to raise the policy above itself and
// strand the retained station configuration without a usable administrator.
IF (Gate = E_GatedAction.ACCESS_POLICY) AND (Level > Access.CurrentLevel) THEN
    RETURN;
END_IF
SetAccessLevel := Access.ConfigureRequired(Gate := Gate, Level := Level);
IF SetAccessLevel THEN
    ConfigRev := ConfigRev + 1;
END_IF
END_METHOD

// §7.7 persistent idle timeout (0 = never), self-gated by ACCESS_POLICY.
METHOD SetSessionTimeout : BOOL
VAR_INPUT
    TimeoutMs : UDINT;
END_VAR
SetSessionTimeout := FALSE;
IF NOT Access.PermitsLogged(Gate := E_GatedAction.ACCESS_POLICY) THEN
    RETURN;
END_IF
SetSessionTimeout := Access.ConfigureSessionTimeout(TimeoutMs := TimeoutMs);
IF SetSessionTimeout THEN
    ConfigRev := ConfigRev + 1;
END_IF
END_METHOD

// §3.8a/§7.7 centralized HMI configuration authority. Concrete overrides never
// need to remember DATA_WRITE or root ownership; they validate only their field.
METHOD WriteConfig : BOOL
VAR_INPUT
    TargetPath : STRING(255);
    WriteKey : STRING(160);
    Revision : DINT;
    TextValue : STRING(255);
END_VAR
WriteConfig := FALSE;
IF (WriteKey = '') OR (Revision <= 0)
OR NOT _M_OwnsModulePath(Path := TargetPath) THEN
    RETURN;
END_IF
// §3.8d - the VALUE's effective write level (its class, raised by its own
// minimum); DATA_WRITE for a value in the built-in class, as before.
IF NOT Access.M_PermitsLevelLogged(Required := _M_DataLevelOf(TargetPath := TargetPath,
        WriteKey := WriteKey, ForWrite := TRUE)) THEN
    RETURN;
END_IF
WriteConfig := _M_WriteBaseConfig(TargetPath := TargetPath, WriteKey := WriteKey,
    Revision := TO_UDINT(Revision), TextValue := TextValue, Commit := TRUE);
IF NOT WriteConfig THEN
    WriteConfig := _M_RouteConfigWrite(TargetPath := TargetPath,
        WriteKey := WriteKey, Revision := TO_UDINT(Revision), TextValue := TextValue);
END_IF
// §3.8a - a model-data value lives in a recipe record too. Another model's edit
// exists ONLY in that record, so failing to save it fails the write; the active
// model's edit is already live, and saving it keeps it across a changeover.
IF WriteConfig AND (TargetPath = Status.Name) AND _M_ModelScopedKey(WriteKey := WriteKey) THEN
    IF NOT _M_SaveModelData() AND (_pModelView <> 0) THEN
        WriteConfig := FALSE;
    END_IF
END_IF
IF WriteConfig THEN
    ConfigRev := ConfigRev + 1;
    _M_MarkPersistPending();           // §3.8b: accepted is LIVE, not yet DURABLE
END_IF
END_METHOD

// §3.8c - the root authority for a capture. Deliberately the same gate, the same
// ownership check and the same ConfigRev bump as WriteConfig: a capture is a
// write whose value came from the machine, and it is no more and no less
// privileged than one the operator typed (§3.8c(d)).
METHOD CaptureConfig : BOOL
VAR_INPUT
    TargetPath : STRING(255);
    WriteKey   : STRING(160);
    Revision   : DINT;
END_VAR
CaptureConfig := FALSE;
IF (WriteKey = '') OR (Revision <= 0)
OR NOT _M_OwnsModulePath(Path := TargetPath) THEN
    RETURN;
END_IF
IF NOT Access.M_PermitsLevelLogged(Required := _M_DataLevelOf(TargetPath := TargetPath,
        WriteKey := WriteKey, ForWrite := TRUE)) THEN
    RETURN;
END_IF
// Framework-owned keys offer no capture: they are policy, not measurements.
CaptureConfig := M_ApplyCapture(Scope := TargetPath, WriteKey := WriteKey,
    Revision := TO_UDINT(Revision), RootReady := (_exec = E_ExecState.READY));
IF CaptureConfig THEN
    ConfigRev := ConfigRev + 1;
END_IF
END_METHOD

// Core §7.5.1 — inject the station's commissioning/engineering gate register at
// Setup, the same shape as SetPartCarrier. Wiring it is what makes the §7.5.2
// standing annunciation appear and what arms the §10.5.1 force surface; a Unit
// with no register is a production Unit and both are simply absent.
//
// Declaring the framework's OWN force gate happens here rather than in the
// project, so a composition root that wires the register cannot forget it
// (§1.1 O1) and cannot arm forcing without also annunciating it.
METHOD SetEngineeringMode
VAR_INPUT
    Mode : REFERENCE TO FB_EngineeringMode;
END_VAR
_engineering REF= Mode;
IF __ISVALIDREF(_engineering) THEN
    _engineering.M_DeclareOutputForcing();
ELSE
    ;
END_IF
END_METHOD

// Core §10.5.1 rules 1 and 3 — may a held force set-point be applied to this
// Unit's outputs right now? The project hardware driver passes the result to
// FB_IoTopologyPublisher.M_ApplyForces every scan, and ForceChannel gates the
// operator request on the identical predicate, so "accepted" and "applied" can
// never disagree. Everything else about a force (access, ownership, direction,
// mapping) is proved elsewhere; this is only the build gate and the mode/state.
METHOD M_ForcePermitted : BOOL
M_ForcePermitted := FALSE;
IF NOT __ISVALIDREF(_engineering) THEN
    RETURN;
END_IF
IF NOT _engineering.ForcingActive THEN
    RETURN;
END_IF
// A running module reasserts its own outputs, so a force is only honest while
// the Unit is idle in MANUAL; leaving either withdraws every force (§10.5.1(3)).
M_ForcePermitted := (_mode = E_Mode.MANUAL) AND (_exec = E_ExecState.READY);
END_METHOD

// Core §7.5.2 — the standing annunciation: one LOW/SYSTEM/AUTO_RESET event per
// registered gate, for as long as that gate is registered.
//
// Why each choice is the way it is, because every one of them is load-bearing:
//   AUTO_RESET  a MANUAL_RESET event refuses Start (§8.3(b)), which would make
//               commissioning gates block the commissioning they exist to serve;
//   LOW/SYSTEM  the lowest priority and the lowest risk class - this says how the
//               software was BUILT, not that the process or safety is impaired,
//               and a louder class would displace real alarms (§8.9);
//   unclearable OperatorReset only closes MANUAL_RESET events, so no operator
//               action reaches this one, and its §8.9 record is not shelvable, so
//               §8.10 cannot silence it either. It closes when the gate is gone -
//               which, gates being build constants, means a new download.
METHOD PRIVATE _M_EngineeringCyclic
VAR
    i : INT;
    gateCount : INT;
END_VAR
IF NOT __ISVALIDREF(_engineering) THEN
    RETURN;
END_IF
gateCount := _engineering.Count;
IF gateCount > PL_Fraktal.MAX_ENGINEERING_GATES THEN
    gateCount := PL_Fraktal.MAX_ENGINEERING_GATES;
END_IF
FOR i := 1 TO gateCount DO
    // Self-healing on purpose. If this slot were ever closed and reused by
    // another event, a remembered index would leave the annunciation silently
    // absent for the rest of the run - the one failure mode a non-clearable
    // message must not have. Re-verify identity, then re-raise.
    IF _engineeringEvt[i] > 0 THEN
        IF (AlarmLog.Active[_engineeringEvt[i]].State = E_AlarmState.CLOSED)
        OR (AlarmLog.Active[_engineeringEvt[i]].ReasonCode <> E_Reason.COMMISSIONING_GATE_ACTIVE) THEN
            _engineeringEvt[i] := 0;
        ELSE
            ;
        END_IF
    ELSE
        ;
    END_IF
    IF _engineeringEvt[i] = 0 THEN
        _engineeringEvt[i] := AlarmLog.Raise(Reason := E_Reason.COMMISSIONING_GATE_ACTIVE,
            Text := _engineering.Gates[i].DescriptionKey, Source := _name,
            Severity := E_Severity.LOW, Category := E_Category.SYSTEM,
            ResetClass := E_ResetClass.AUTO_RESET);
    ELSE
        ;
    END_IF
END_FOR
END_METHOD

// §10.5.1 centralized force authority. Only an idle MANUAL Unit may reach the
// application resolver; that resolver still proves root ownership, OUTPUT,
// non-safety identity, mapping and the channel-specific release.
METHOD ForceChannel : BOOL
VAR_INPUT
    ChannelPath : STRING(255);
    Force : BOOL;
    BoolText : STRING(255);
    AnalogText : STRING(160);
END_VAR
ForceChannel := FALSE;
IF NOT Access.PermitsLogged(Gate := E_GatedAction.MANUAL) THEN
    RETURN;
END_IF
// §10.5.1 rules 1 and 3 in one predicate, the same one the hardware driver
// applies each scan - so the request can never be accepted under conditions
// under which the force would not actually be applied.
IF NOT M_ForcePermitted() OR (ChannelPath = '') THEN
    RETURN;
END_IF
ForceChannel := _M_RouteForceChannel(ChannelPath := ChannelPath, Force := Force,
    BoolText := BoolText, AnalogText := AnalogText);
END_METHOD

// Core §7.8 — full rollup for the simpler gated Unit actions (Stop, ALARM_RESET,
// CHANGEOVER, MODE_CHANGE, step). Same predicate the gates use. Start has its own
// richer ReleaseReportStart (interlocks); manual has ReleaseReportManual (target).
METHOD ReleaseReportAction : BOOL
VAR_INPUT
    Gate : E_GatedAction;
END_VAR
VAR_IN_OUT
    Report : ST_ReleaseReport;
END_VAR
Report.Count := 0;
Report.Released := FALSE;
// access is the common gate
IF NOT Access.Permits(Gate := Gate) THEN
    _M_AddReason(Report := Report, Text := 'std.release.insufficientAction', Reason := E_Reason.NONE, Kind := E_ReleaseKind.ACCESS);
END_IF
// per-action state preconditions
CASE Gate OF
    E_GatedAction.CHANGEOVER:
        IF _exec = E_ExecState.BUSY THEN
            _M_AddReason(Report := Report, Text := 'std.release.changeoverRunning', Reason := E_Reason.NONE, Kind := E_ReleaseKind.MODE);
        END_IF
    E_GatedAction.ALARM_RESET:
        IF NOT AlarmLog.Blocking THEN
            _M_AddReason(Report := Report, Text := 'std.release.noBlockingAlarm', Reason := E_Reason.NONE, Kind := E_ReleaseKind.OTHER);
        END_IF
    E_GatedAction.MODE_CHANGE:
        IF _modePend THEN
            _M_AddReason(Report := Report, Text := 'std.release.modeChangeAlreadyPending', Reason := E_Reason.NONE, Kind := E_ReleaseKind.MODE);
        ELSIF (_exec = E_ExecState.BUSY)
        AND (ModePolicy[TO_INT(_mode)].Shield = E_ModeSwitchShield.BLOCKED_WHILE_RUNNING) THEN
            _M_AddReason(Report := Report, Text := 'std.release.modeSwitchBlockedWhileRunning',
                Reason := E_Reason.NONE, Kind := E_ReleaseKind.MODE);
        ELSE
            ;
        END_IF
ELSE
    ;                                          // actions with no extra state predicate
END_CASE
Report.Released := (Report.Count = 0);
ReleaseReportAction := Report.Released;
END_METHOD

// Core §7.8 — full rollup of why a manual command to Target would be refused (§7.6.1).
METHOD ReleaseReportManual : BOOL
VAR_INPUT
    TargetPath : STRING(255);
    Value : DINT;
END_VAR
VAR_IN_OUT
    Report : ST_ReleaseReport;
END_VAR
Report.Count := 0;
Report.Released := FALSE;
IF _mode <> E_Mode.MANUAL THEN
    _M_AddReason(Report := Report, Text := 'std.release.manualModeRequired', Reason := E_Reason.NONE, Kind := E_ReleaseKind.MODE);
END_IF
IF NOT Access.Permits(Gate := E_GatedAction.MANUAL) THEN
    _M_AddReason(Report := Report, Text := 'std.release.insufficientManual', Reason := E_Reason.NONE, Kind := E_ReleaseKind.ACCESS);
END_IF
_M_AppendManualInterlocks(TargetPath := TargetPath, Value := Value, Report := Report);  // §7.6, target+command-aware
Report.Released := (Report.Count = 0);
ReleaseReportManual := Report.Released;
END_METHOD

// Core §7.8 — pure query: the FULL rollup of why Start would be refused right now.
// This is the authoritative machine predicate consumed by Start (no drift).
// Released = TRUE means Start proceeds. Lists mode + access + blocking-alarm,
// control-domain, and concrete mode-entry release reasons. The caller owns the
// bounded report storage; returning this large record by value can overflow a
// TwinCAT task stack when Start consumes the result.
METHOD ReleaseReportStart : BOOL
VAR_IN_OUT
    Report : ST_ReleaseReport;
END_VAR
Report.Count := 0;
Report.Released := FALSE;
// access (§7.7)
IF NOT Access.Permits(Gate := E_GatedAction.START_STOP) THEN
    _M_AddReason(Report := Report, Text := 'std.release.insufficientStartStop', Reason := E_Reason.NONE, Kind := E_ReleaseKind.ACCESS);
END_IF
// mode / run state (§3.4)
IF _modePend THEN
    _M_AddReason(Report := Report, Text := 'std.release.modeChangePending', Reason := E_Reason.NONE, Kind := E_ReleaseKind.MODE);
END_IF
IF _mode = E_Mode.MANUAL THEN
    _M_AddReason(Report := Report, Text := 'std.release.manualHasNoAutoSequence', Reason := E_Reason.NONE, Kind := E_ReleaseKind.MODE);
END_IF
IF _exec <> E_ExecState.READY THEN
    _M_AddReason(Report := Report, Text := 'std.release.unitNotReady', Reason := E_Reason.NONE, Kind := E_ReleaseKind.MODE);
END_IF
// blocking alarm (§8.3)
IF AlarmLog.Blocking THEN
    _M_AddReason(Report := Report, Text := 'std.release.manualReset', Reason := E_Reason.NONE, Kind := E_ReleaseKind.ALARM);
END_IF
// lost configuration image (§3.8b): the DEPLOYMENT's declared consequence. The
// policy was stored and published but read nowhere, so a station that declared
// BLOCK_UNTIL_ACKNOWLEDGED started on defaults anyway. This is where it is read.
IF ConfigPersist.RestoreLost AND NOT ConfigPersist.RestoreAcknowledged
AND (ConfigPersist.RestorePolicy = E_ConfigRestorePolicy.BLOCK_UNTIL_ACKNOWLEDGED) THEN
    _M_AddReason(Report := Report, Text := 'std.release.configRestoreUnacknowledged', Reason := E_Reason.CONFIG_RESTORE_LOST, Kind := E_ReleaseKind.ALARM);
END_IF
IF ControlDomain.Present AND NOT ControlDomain.ReadyForStart THEN
    _M_AddReason(Report := Report, Text := 'std.release.controlDomainNotReady', Reason := E_Reason.NONE, Kind := E_ReleaseKind.INTERLOCK);
END_IF
// active mode's immediate entry/frontier conditions (concrete override)
_M_AppendInterlocks(Report := Report);
Report.Released := (Report.Count = 0);
ReleaseReportStart := Report.Released;
END_METHOD

// §8.5.1 — clear accumulators + ring (shift start). Gated: §7.7 DATA_WRITE; audited §8.3.
METHOD ResetOee : BOOL
VAR
    i : INT;
    auditSlot : INT;
END_VAR
IF NOT Access.PermitsLogged(Gate := E_GatedAction.DATA_WRITE) THEN
    ResetOee := FALSE;
    RETURN;
END_IF
Oee.RunMs := 0; Oee.DownMs := 0; Oee.IdleMs := 0;
FOR i := 1 TO PL_Fraktal.MAX_OEE_SAMPLES DO
    OeeTrend[i].Oee := 0.0; OeeTrend[i].OeeValid := FALSE;
    OeeTrend[i].Availability := 0.0; OeeTrend[i].Performance := 0.0; OeeTrend[i].Quality := 0.0;
END_FOR
OeeTrendHead := 0;
_oeeSampMs := 0;
_M_OeeCompute();
_shiftManualReset := TRUE;                  // §8.5.2(c): the shift record will say so
auditSlot := AlarmLog.Raise(Reason := E_Reason.NONE,
    Text := 'std.audit.oeeReset', Source := _name,
    Severity := E_Severity.LOW, Category := E_Category.SYSTEM, ResetClass := E_ResetClass.AUTO_RESET);
IF auditSlot > 0 THEN AlarmLog.Gone(Slot := auditSlot); END_IF
ResetOee := TRUE;
END_METHOD

// §3.4.2 — HMI HOLD_TO_RUN input. NON-SAFETY (§9): never a dead-man; interlocks
// still apply at every step. TRUE only while the operator holds the button.
METHOD SetHoldRun : BOOL
VAR_INPUT
    Held : BOOL;
END_VAR
IF Held AND (NOT Access.PermitsLogged(Gate := E_GatedAction.START_STOP)
OR (RunStyle <> E_RunStyle.HOLD_TO_RUN) OR (_exec <> E_ExecState.BUSY)) THEN
    SetHoldRun := FALSE;
    RETURN;
END_IF
_holdRun := Held;                     // FALSE is always accepted so a hold cannot stick
SetHoldRun := TRUE;
END_METHOD

// §8.5.1 — configure the ideal cycle time (per model, §3.8). 0 disables Performance.
METHOD SetIdealCycle : BOOL
VAR_INPUT
    Ms : UDINT;
END_VAR
Oee.IdealCycleMs := Ms;
SetIdealCycle := TRUE;
END_METHOD

// §3.4/§3.7 — FALSE = unsupported (graceful rejection); TRUE = committed or pending
METHOD SetMode : BOOL
VAR_INPUT
    Mode : E_Mode;
END_VAR
IF NOT Access.PermitsLogged(Gate := E_GatedAction.MODE_CHANGE) THEN
    SetMode := FALSE;                  // §7.7(c): who-gate ANDs the machine gates
    RETURN;
END_IF
IF NOT _M_Supports(Mode) THEN
    SetMode := FALSE;
    RETURN;
END_IF
IF (Mode = _mode) AND NOT _modePend THEN
    SetMode := TRUE;
    RETURN;
END_IF
// §3.4.1 shield: policy of the mode being LEFT governs while its sequence runs
IF (_exec = E_ExecState.BUSY)
AND (ModePolicy[TO_INT(_mode)].Shield = E_ModeSwitchShield.BLOCKED_WHILE_RUNNING) THEN
    SetMode := FALSE;                  // must Stop first (graceful rejection, not a fault)
    RETURN;
END_IF
IF (NOT _modePend) OR (_modeReq <> Mode) THEN
    _modeExitFirst := TRUE;
END_IF
_modeReq := Mode;
_modePend := TRUE;
SetMode := TRUE;
END_METHOD

// §3.1b/§3.8 — transactional model change: prepare the whole subtree, then commit.
METHOD SetModel : BOOL
VAR_INPUT
    Id : ST_ModelId;
END_VAR
IF NOT Access.PermitsLogged(Gate := E_GatedAction.CHANGEOVER) THEN
    SetModel := FALSE;                 // §7.7
    RETURN;
END_IF
IF _exec = E_ExecState.BUSY THEN
    SetModel := FALSE;                 // changeover is not mid-cycle (§3.8 loads at CHANGEOVER)
    RETURN;
END_IF
IF NOT PrepareRecipe(Model := Id) THEN
    AbortRecipe();
    SetModel := FALSE;
    RETURN;
END_IF
CommitRecipe();                         // infallible after successful preparation
Model := Id;                           // identity changes only after subtree commit
ConfigRev := ConfigRev + 1;            // §3.10.2 — recipe/config leaves changed
SetModel := TRUE;
END_METHOD

// §11.6.1 internal composition seam; not a remote command surface.
METHOD M_PublishMaterialChanged : BOOL
VAR_INPUT
    Material : STRING(80);
    Value    : STRING(80);
END_VAR
M_PublishMaterialChanged := _M_HostEvent(
    Kind := E_HostEventKind.MATERIAL_CHANGED, PartUid := '', Subject := Material,
    Value := Value, Verdict := E_Verdict.NONE, ReasonCode := E_Reason.NONE);
END_METHOD

// §11.6.1 internal composition seam; not a remote command surface.
METHOD M_PublishToolChanged : BOOL
VAR_INPUT
    Tool  : STRING(80);
    Value : STRING(80);
END_VAR
M_PublishToolChanged := _M_HostEvent(
    Kind := E_HostEventKind.TOOL_CHANGED, PartUid := '', Subject := Tool,
    Value := Value, Verdict := E_Verdict.NONE, ReasonCode := E_Reason.NONE);
END_METHOD

// §11.6.2 inject an optional OPC UA/MES/REST/MQTT delivery adapter.
METHOD M_SetHostEventSink : BOOL
VAR_INPUT
    Sink : I_HostEventSink;
END_VAR
M_SetHostEventSink := HostEvents.SetSink(Sink := Sink);
END_METHOD

// §3.16.2 — inject the part carrier at the composition root (0 = traceability off).
// Source-agnostic: BY_POSITION local, RFID, DataMatrix, or host, behind I_PartCarrier.
METHOD SetPartCarrier : BOOL
VAR_INPUT
    Carrier : I_PartCarrier;
END_VAR
_carrier := Carrier;
SetPartCarrier := (Carrier <> 0);
END_METHOD

// §3.4.2 — HMI selects the run style for the active mode. Modes that don't opt in
// (see _M_SupportsRunStyle) reject non-CONTINUOUS. Access: MODE_CHANGE-gated (§7.7).
METHOD SetRunStyle : BOOL
VAR_INPUT
    Style : E_RunStyle;
END_VAR
IF NOT Access.PermitsLogged(Gate := E_GatedAction.MODE_CHANGE) THEN
    SetRunStyle := FALSE;
    RETURN;
END_IF
IF (Style <> E_RunStyle.CONTINUOUS) AND NOT _M_SupportsRunStyle(Style := Style) THEN
    SetRunStyle := FALSE;               // mode didn't opt into stepping (graceful reject)
    RETURN;
END_IF
RunStyle := Style;
SetRunStyle := TRUE;
END_METHOD

// §8.10 — gated HMI entry: shelve an active alarm's ANNUNCIATION (control untouched).
// §7.7 ALARM_SHELVE + audit; refuses SAFETY / unrationalized reasons (AlarmLog rules).
METHOD ShelveAlarm : BOOL
VAR_INPUT
    Slot      : INT;
    DurationS : UDINT;
END_VAR
IF NOT Access.PermitsLogged(Gate := E_GatedAction.ALARM_SHELVE) THEN
    ShelveAlarm := FALSE;
    RETURN;
END_IF
ShelveAlarm := AlarmLog.Shelve(Slot := Slot, DurationS := DurationS);
END_METHOD

// §3.3/§6 intro — the run IS a §6.1 command.
// §7.8: ReleaseReportStart is the authoritative machine gate as well as the
// operator explanation, so a concrete Unit cannot report an interlock it ignores.
// Build directly into the published response storage: ST_ReleaseReport is too
// large for nested by-value/local copies on a small TwinCAT task stack.
METHOD Start : BOOL
IF NOT Access.PermitsLogged(Gate := E_GatedAction.START_STOP) THEN
    Start := FALSE;                    // §7.7
    RETURN;
END_IF
IF ReleaseReportStart(Report := HmiResponse.Report) THEN
    _stopReq := FALSE;                 // §8.3(b): a MANUAL_RESET event blocks restart
    Execute := TRUE;
    Start := TRUE;
ELSE
    Start := FALSE;
END_IF
END_METHOD

// §3.4.2 — HMI single-step: request advance of one step (edge-consumed by _M_StepGate).
METHOD StepRequest : BOOL
IF NOT Access.PermitsLogged(Gate := E_GatedAction.START_STOP)
OR (RunStyle <> E_RunStyle.SINGLE_STEP) OR (_exec <> E_ExecState.BUSY) THEN
    StepRequest := FALSE;
    RETURN;
END_IF
_stepReq := TRUE;
StepRequest := TRUE;
END_METHOD

// §3.3 — stop after the current cycle
METHOD Stop : BOOL
IF NOT Access.PermitsLogged(Gate := E_GatedAction.START_STOP) THEN
    Stop := FALSE;                     // §7.7
    RETURN;
END_IF
IF _exec = E_ExecState.BUSY THEN
    _stopReq := TRUE;
ELSE
    _stopReq := FALSE;
    Execute := FALSE;                  // release a terminal run command (ERROR/DONE/ABORTED)
END_IF
Stop := TRUE;
END_METHOD

// §3.4 — TRUE while a stop is requested but the sequence is still finishing
// (running -> stopping). HMI blinks the stop button on this.
PROPERTY StopPending : BOOL
GET
StopPending := _stopReq AND (_exec = E_ExecState.BUSY);
END_GET
END_PROPERTY

// §8.10 — gated HMI entry: restore annunciation.
METHOD UnshelveAlarm : BOOL
VAR_INPUT
    Slot : INT;
END_VAR
IF NOT Access.PermitsLogged(Gate := E_GatedAction.ALARM_SHELVE) THEN
    UnshelveAlarm := FALSE;
    RETURN;
END_IF
UnshelveAlarm := AlarmLog.Unshelve(Slot := Slot);
END_METHOD

END_FUNCTION_BLOCK

(* stored: Version 1.1.0.1, ProductVersion 3.1.4024.16
   POU FB_UnitBase: Id {116d9026-fbad-4cf8-8b52-50d17613c706}, SpecialFunc None
   Method _M_AddReason: Id {63c5e93f-708a-4c3a-aa1b-ee43d815fb4a}
   Method _M_AppendInterlocks: Id {2bc971ff-4cee-49e6-a29f-4f727818205b}
   Method _M_AppendManualInterlocks: Id {c18caeb9-871a-4a4c-aad2-2711e3ced37a}
   Method _M_AppendDecisionInterlocks: Id {bbac41d9-35ba-4800-af52-51cd30b49db7}
   Method _M_AskDecision: Id {4e23ce8a-174c-4663-9cbe-be702ba37032}
   Method _M_ClearDecisionState: Id {db09e3d9-4427-4607-8a90-66b39812e37b}
   Method _M_DecisionCyclic: Id {ff058255-d664-4ce3-986d-8ad7a970388c}
   Method _M_DecisionMatches: Id {2ca48458-620f-4a17-b6d1-b5680778bd4e}
   Method _M_LogDecision: Id {eb357477-2029-4b6d-8688-04dc5df5e04b}
   Method _M_ValidateDecision: Id {1229fbc9-7dc8-4907-b878-f6af733f2c09}
   Method _M_Await: Id {098638cb-fc78-4032-9954-0ceffe6b565c}
   Method _M_CascadeMode: Id {3ac20481-72c5-4cd1-88e5-b9f7eb433162}
   Method _M_ClearPending: Id {cb01b1f4-f591-43f7-a826-970be7300b04}
   Method _M_AuditHmiAccepted: Id {f8865f87-3ae7-472e-b775-3408513a4586}
   Method _M_OwnsModulePath: Id {9b8c6045-f404-4484-937e-b0a8f749d8fd}
   Method _M_EndOfCycle: Id {9824e487-d8d3-4cb9-8c78-a6d2fc09a62d}
   Method _M_HandleHmiRequest: Id {63ae9d50-339f-4904-a8ec-81f853aed962}
   Method _M_HostEvent: Id {76fb49ac-f9ea-4e53-8db6-e7e4e756fd84}
   Method _M_InitModePolicy: Id {df8ba8da-c8fa-411c-85c1-392b353d5cfd}
   Method _M_OeeCompute: Id {2991f1a8-70f1-48a9-aa83-352243818d0a}
   Method _M_OeeUpdate: Id {8a4f011d-5d7a-4935-ad26-8a5fbcf63643}
   Method _M_PartAborted: Id {a55c31e8-06f9-4d10-8c26-4e83b7d5c1f2}
   Method _M_PartEvent: Id {f18c2d47-9b53-4e6a-8c02-3a71d5f0b429}
   Method _M_PartProcessed: Id {e91b5a02-73df-4f16-a8d4-1c30fe8a97d2}
   Method _M_PartReceived: Id {58c0a7d9-14be-4f22-8d6a-9b2ef4c1e370}
   Method _M_PartRecord: Id {7be4f6a3-1d20-4c8e-be55-f2a09318d67c}
   Method _M_PartStarted: Id {02a97d1c-6bb5-4f80-9d34-c58b12f04ae6}
   Method _M_PublishStatus: Id {02d44270-09e8-4bc1-97fd-f43dd3fc44f2}
   Method _M_PushHistory: Id {3f9af757-7ef5-4499-8b8d-04dcd97acc93}
   Method _M_RaiseMaintenance: Id {c92e4b71-6d05-4f88-9e3a-2b17d4c8a054}
   Method _M_RouteConfigWrite: Id {4e524daf-e482-4764-8639-e58c1f363aa3}
   Method _M_WriteBaseConfig: Id {c30f39b4-eae4-421d-a415-c6dc3b402679}
   Method _M_RouteForceChannel: Id {301182d5-8822-451a-950c-49d23daf4640}
   Method _M_RouteManual: Id {9fa4e2c2-3f5f-4681-aed5-559f1df0d2c6}
   Method _M_RecordSequenceStep: Id {bae7334e-b67d-46db-a917-aa05f1522e0f}
   Method _M_ResetSequenceRows: Id {3a7e979a-9c02-4e58-aa36-f0627902f8fb}
   Method _M_SequenceAnnotate: Id {981fa92c-f12b-4972-9483-880edfae72c8}
   Method _M_SequenceAnnotationClear: Id {7256d50d-cf16-4906-8e35-fd394563602f}
   Method _M_SetStep: Id {1066dd3c-baf2-43ea-91d5-309ad4ca7878}
   Method _M_StallWalk: Id {ee453cd4-7027-4207-b43e-f1a12367922c}
   Method _M_StepGate: Id {853d1e75-22c1-46fb-9a92-007882839a98}
   Method _M_Supports: Id {5285aa9e-3e18-4090-bed9-0119293228bb}
   Method _M_SupportsRunStyle: Id {f4e81ed4-d8b0-494c-bd7a-6b417d6219cf}
   Method _M_TakeDecision: Id {e2e1443d-0421-4608-8ae5-b7bb44177b3c}
   Method CountGood: Id {852e951b-039f-45bd-80a3-6417310e2406}
   Method CountNok: Id {a686f5b6-4c90-4e12-9d98-fa111d14dfe8}
   Method CountRework: Id {5c8e02d7-9a41-4f36-8b52-e04a71c6d983}
   Method M_AppendConfig: Id {29c7f5d4-0b81-4ae3-9762-84f6d013ba58}
   Method SetConfigStore: Id {1f6b90d4-38a2-4c57-9e01-b47d2c85a3f6}
   Method SetConfigPersistence: Id {a5c37e08-9412-4bd6-83f9-6e05b17c94a2}
   Method SetConfigPersistWindow: Id {5db2740a-9e18-4c63-b0f5-8a2914e7c036}
   Method SetConfigRestorePolicy: Id {72e4a1b9-c530-46df-8127-93b605ea4d78}
   Method _M_MarkPersistPending: Id {6d09fb35-2a84-41ce-b7f0-58d2e1937a4b}
   Method _M_ConfigPersistFailed: Id {3a81c6e7-40b2-4d95-916f-c82705bd4e13}
   Method _M_ConfigPersistCyclic: Id {9c0d4318-b7a5-42e6-8f13-05ea7c9b2d40}
   Method _M_DrainRestoreLoss: Id {0b7e5294-16ad-43c1-a8f6-249d038be715}
   Method AcknowledgeConfigRestore: Id {e18c47b3-5029-4ed6-9a71-b3406fc25d89}
   Method _M_RejectConfigSet: Id {5f2a90c6-8b41-4d73-bec0-172e845f39ab}
   Method _M_SetOpAllowed: Id {3d70b95e-c284-41f0-86ba-9e15c703da42}
   Method DeleteConfigSet: Id {e533f05f-2594-42e8-8c99-81d549fc4090}
   Method _M_DataLevelOf: Id {181e4912-d325-4208-982a-bde235412443}
   Method M_DeclareDataClass: Id {b9a4a5ae-9fab-42bd-bc82-7e32dffbd2a9}
   Method SetDataClassLevel: Id {047e7f36-274a-4350-8ad6-b77d4f72cc43}
   Method _M_IsLineKey: Id {59358b2d-9028-416d-b8b1-1699a6cd425f}
   Method M_ApplyConfigWrite: Id {09d95f4a-6281-4745-bbd6-78a379c3dcc0}
   Method M_StageConfigWrite: Id {c033d610-c896-4206-a3ad-81018a4dd465}
   Method M_ApplyCapture: Id {e2ff8450-6122-448e-b867-574b3000edfa}
   Method M_ConfigAccessOf: Id {b5882f05-b837-4f44-ba08-a65bdacad4e2}
   Method M_RegisterModelData: Id {9e19e4d6-5131-4b98-84c6-f84c0e107ced}
   Method _M_OpenModelView: Id {93ccf92c-d752-48c8-af0b-7941488b3430}
   Method WriteModelConfig: Id {2a0d9e3e-ba70-4e09-955f-cec98e39642e}
   Method M_AppendModelConfig: Id {0e6d90bf-ad76-4384-ab12-1767af3d1a4f}
   Method _M_SaveModelData: Id {614f64a8-a7bb-415b-89b6-cd5638516728}
   Method SetLine: Id {b3e3c826-6085-43fe-ab9e-5ee8d63ca7f0}
   Method M_ShiftTick: Id {4606cb81-948b-4fb3-a998-828e0341cdfd}
   Method _M_CloseShift: Id {3589014a-a797-47c8-9c22-164193338f8a}
   Method SaveConfigSet: Id {8a4d1e07-63b9-4c25-90fd-e7285a1cb046}
   Method LoadConfigSet: Id {c93f5b28-047e-41da-b6c1-5820ae74f3d9}
   Method _M_StageOneRecord: Id {b6014e8d-72c3-49a5-80fe-c1738d92406b}
   Method _M_ConfigSetHalfApplied: Id {47db6015-9a2e-4c38-b7f0-d5216e409a83}
   Method ListConfigSets: Id {2e85d740-c6b1-4930-a5df-08417b3ce629}
   Method ExportConfigSetLine: Id {6c1908fe-b432-4a07-95d8-e2603ba7145c}
   Method ImportConfigSetLine: Id {d0a76321-8e54-4bc9-97a2-3f16054eb7d8}
   Method ImportConfigSetPiece: Id {fe4a451b-e9cc-440c-9ade-c56031168c94}
   Method M_SequenceAskDecision: Id {099b4f9d-bc09-44d1-a376-b2e504dbb242}
   Method M_SequenceAwait: Id {c61669f7-ff2f-475c-915e-c23e673ae50d}
   Method M_SequenceClearDecision: Id {f5e88d63-dd7e-45c7-8fcc-149437ebcb66}
   Method M_SequenceComplete: Id {94f85c2c-bf7e-4679-9ad7-df299f9443e9}
   Method M_SequenceCountGood: Id {7ac5d064-bbc3-4e23-a999-5b1106c18501}
   Method M_SequenceEndOfCycle: Id {2465831e-ce6a-49ba-894a-d94a6e5b730d}
   Method M_SequenceFault: Id {6dcf30ea-273a-4919-b53c-93ee346a0722}
   Method M_SequencePartProcessed: Id {f3fe635f-f0ef-4b80-918f-2af11c08a018}
   Method M_SequencePartReceived: Id {9576ad5e-fef2-4d71-bd9f-075e2fbf7f48}
   Method M_SequencePartRecord: Id {272bc8d6-51f1-4e02-a0f6-834fc34cf443}
   Method M_SequencePartStarted: Id {c34399dc-9677-414b-87a7-da41fec81ce1}
   Method M_SequenceRegister: Id {9c12e1e0-2b54-4710-a719-b7dbb939da2c}
   Method _M_BeginSequenceScan: Id {90d173ad-1ac7-44ea-8963-773d827fd02e}
   Method _M_RestartSequences: Id {a7179c76-6bab-4060-a5d3-1d37fa9ff028}
   Method OnAbort: Id {045fbfe7-105f-49b4-bf25-f60661612052}
   Method OnAbortInError: Id {f7465218-0d83-46fd-a26a-73b938ae69a7}
   Method M_SequenceWarn: Id {75ce463f-f749-4a05-8c5e-fea3607d380d}
   Method M_SequenceRaise: Id {0bee2dd9-d8a8-4946-b400-dc31452b748f}
   Method _M_ResumeSequencesAfterError: Id {f331535e-fb67-4439-a403-97a206176d31}
   Method M_SequenceSetStep: Id {cd33b52b-b93d-4827-921b-0507be840f66}
   Method M_SequenceStepGate: Id {4300b99e-dada-4558-9a7d-f357bb3b59db}
   Method M_SequenceStopNow: Id {5e2a91d7-38c4-4b0f-a6e8-74d19c2b50f3}
   Method M_SequenceStopPending: Id {9b04e7c1-52d8-4f36-8a92-1c65fd83a247}
   Method M_SequenceTakeDecision: Id {a0cad3a5-90f7-4b63-9dfc-d75845d8e702}
   Method ManualHeldTo: Id {9a41c8e0-5b73-4d26-81fa-06e5327d94b1}
   Method _M_RouteHeld: Id {3c78e05b-1246-4a9d-b0e7-52f8146c93da}
   Method _M_ChartRevCyclic: Id {b40f7e26-95a1-4d83-b217-0c6e59a71e34}
   Method _M_HeldCyclic: Id {d51937ae-64c2-408f-9b13-27e0a4586cf7}
   Method ManualCommandTo: Id {4de99325-2725-4710-8292-b2f11cd5c61c}
   Property ModeActive: Id {cadd011f-36e9-480f-9687-f764db6a93a1}
   Get Get: Id {480f723e-9802-4414-9cf5-b9bf28538b7e}
   Property ModelCode: Id {52be901d-358c-42d1-8de9-24cabf037285}
   Get Get: Id {d1228112-dc00-4a78-8d96-06a0aa3db5e2}
   Property ModuleType: Id {19c4f994-fbe0-4e50-80d5-d89b1a1fb1fa}
   Get Get: Id {e694d09e-29b1-48cc-b1e6-0d26ae208150}
   Method OnCyclic: Id {833bee58-3464-412f-8fa3-37fa398fef55}
   Method _M_HighestSeverity: Id {06beeb70-94f2-4095-9daa-a1af1fd36a20}
   Method RequestLampTest: Id {0a1df30a-092c-4f3f-91a5-1af799e7cb11}
   Method SetSignalTowerConfig: Id {93bf4461-f32d-446c-ac46-8d0b800f56d9}
   Method SetSystemHealth: Id {f544458e-b3ee-4aad-ac8d-2565c5120fa3}
   Method OnInit: Id {c11afaa2-3957-4d40-8695-293ff272dfc1}
   Method OnModeChanged: Id {4307796c-f352-4515-b104-1671ef41b10c}
   Method OnCommandStart: Id {4698d7ce-6d4c-492c-9ead-e072c285ae34}
   Method OnModeExit: Id {d824838b-6d6c-4575-ade3-00f3815d6c9e}
   Method OperatorReset: Id {86e0365e-0665-41e9-b6f4-1156fe1cf971}
   Method _M_RecoverState: Id {2d0b998f-abd6-473c-8cb5-b6b35c39d09a}
   Method OnOperatorReset: Id {ad173c6c-fa19-47ee-a347-f5b5e0c7654a}
   Method RequestLocalReset: Id {2ac5c84b-a29d-437a-b5c9-0d4b5d278812}
   Method RegisterAvailableModel: Id {651bb1e1-71c6-4fb4-a063-4ea057e752cf}
   Method RequestControlPower: Id {cb696b98-d3f2-48ed-8f23-09e45169ea5f}
   Method SubmitDecision: Id {70347f2b-2424-4514-beb7-8788c8d00fca}
   Method SetAccessLevel: Id {a2b5995c-ea0a-4911-83f3-0a5e24269563}
   Method SetSessionTimeout: Id {e8244b36-18c3-4b2a-8ef7-db39a1dfa257}
   Method WriteConfig: Id {3e40e571-e45f-4204-a5d3-c9907077e8b2}
   Method CaptureConfig: Id {6657c29b-54a9-410f-b368-d4a1ad1bb646}
   Method SetEngineeringMode: Id {28e702f3-e7d8-4e5a-8206-7208a16b6696}
   Method M_ForcePermitted: Id {b9d8bf79-0c6d-4741-99f8-f427bda243e9}
   Method _M_EngineeringCyclic: Id {0b6876ea-bb0c-4e77-ab09-61eab13a8627}
   Method ForceChannel: Id {8bf9fd9d-8084-4dbf-b41b-c60e5e0cc995}
   Method ReleaseReportAction: Id {b52c134c-be50-4c5c-b4df-ad025ff72931}
   Method ReleaseReportManual: Id {9e9f491d-e5a8-435c-bc95-8f93e8c3530b}
   Method ReleaseReportStart: Id {c78c7568-83f2-4d9d-9ae3-f47850cbc022}
   Method ResetOee: Id {76d2024b-e4e9-424e-bbf4-fcfd488c8439}
   Method SetHoldRun: Id {fbc37d38-8939-4f18-83b4-eb1341e2b47b}
   Method SetIdealCycle: Id {21a43259-c0d5-420f-993f-704ffad3d187}
   Method SetMode: Id {7da8ba28-e926-421f-9272-a6c57a552866}
   Method SetModel: Id {6a7ae71f-5111-44b3-bfc5-fd8bfdcd3719}
   Method M_PublishMaterialChanged: Id {27225091-fd15-48c0-a242-131de64ab93c}
   Method M_PublishToolChanged: Id {cc18bd59-d3df-4af3-a8b4-e56788466431}
   Method M_SetHostEventSink: Id {c075ef1c-ce1a-4aec-9cd4-f8cc578ba7b2}
   Method SetPartCarrier: Id {6a3e9c15-2f84-4b0d-9c17-d84f5e21ab63}
   Method SetRunStyle: Id {f598b9ad-9cb8-47de-920d-91798ab2094a}
   Method ShelveAlarm: Id {254b8716-80f2-462f-8e49-d89ea86b5224}
   Method Start: Id {cf23e563-6a38-441b-bf71-cf054a5930b3}
   Method StepRequest: Id {64e64e1a-0c5a-460b-882a-ab14da4420e6}
   Method Stop: Id {a7c9b0f8-857c-458d-afc6-9746ac288208}
   Property StopPending: Id {f114fa1a-de45-4aa0-be5b-cf63c773b8b7}
   Get Get: Id {135b3f46-0e90-48aa-8ac1-6493d51adeb3}
   Method UnshelveAlarm: Id {f39e65ca-0fee-42d8-be9a-7e2098b02e14} *)
